{attribute 'qualified_only'}
VAR_GLOBAL
	Rotor_X: INT;
	Rotor_Y: INT;
	Rotor_Z: INT;
END_VAR

(* stored: Version 1.1.0.1, ProductVersion 3.1.4024.4
   GVL GVL: Id {5accb902-7e9e-45d7-8000-bd24352e736f} *)
